// TIA Portal V16 export
// export: Created 2021-07-12T14:47:18.6278253Z, ExportSetting WithDefaults, DisplayName Totally Integrated Automation Portal, DisplayVersion V16, DisplayName TIA Portal Version Control Interface, DisplayVersion V16, DisplayName TIA Portal Openness, DisplayVersion V16, DisplayName STEP 7 Professional, DisplayVersion V16, DisplayName STEP 7 Safety, DisplayVersion V16, DisplayName WinCC Professional, DisplayVersion V16
TYPE "LSimaHydTO_typeTransducer"
TITLE = LSimaHydTO_typeTransducer
// Pressure transducer configuration
// stored: IsFailsafeCompliant false
   STRUCT
      HWReference { S7_SetPoint := 'True'} : Int := 16#6C00;   // Normalization of the raw value for 100%. Distinction between a SIMATIC or a SINAMICS periphery: SIMATIC = 27648, SINAMICS = 16384
      NominalPressure { S7_SetPoint := 'True'} : LReal := 400.0;   // Nominal pressure of transducer, e.g. 400 [bar]
      Area { S7_SetPoint := 'True'} : LReal := 1.0;   // Area [mm2] or [in2]
      Offset { S7_SetPoint := 'True'} : LReal := 0.0;   // Offset in pressure units
      FilterTime { S7_SetPoint := 'True'} : LReal := 0.0;   // Smoothing filter
      ErrorValue { S7_SetPoint := 'True'} : Word := 16#7FFF;   // Error signal
   END_STRUCT;
END_TYPE
